FUNCTION TryConvert_UINT_TO_USINT : BOOL
VAR_INPUT
	in : UINT;
	out : REFERENCE TO USINT;
END_VAR

IF in > DatatypeLimits.MAX_VALUE_OF_UINT_WHICH_CAN_BE_HELD_IN_A_USINT THEN
	RETURN;
END_IF

out := UINT_TO_USINT(in);
TryConvert_UINT_TO_USINT := TRUE;

END_FUNCTION

(* stored: Version 1.1.0.1, ProductVersion 3.1.4024.12
   POU TryConvert_UINT_TO_USINT: Id {c5542c81-bd92-4584-a70e-e87ca1ac518e}, SpecialFunc None *)
